Omron CX-Programmer project NewProject (CX-Programmer 9.61)

# PLC NewPLC1: CJ1M CPU11

## Global symbols (name address type ; comment)
0.00 BOOL  ; PB_Start
0.01 BOOL  ; PB_Stop
10.00 BOOL  ; IR_Control
10.01 BOOL  ; SIMPANG 1 = HIJAU
10.02 BOOL  ; SIMPANG 1 = KUNING
10.03 BOOL  ; SIMPANG1 = MERAH
10.04 BOOL  ; SIMPANG 2= HIJAU
10.05 BOOL  ; SIMPANG 2 = KUNING
10.06 BOOL  ; SIMPANG 2 = MERAH
10.07 BOOL  ; SIMPANG 3 = HIJAU
10.08 BOOL  ; SIMPANG 3 = KUNING
10.09 BOOL  ; SIMPANG 3 = MERAH
10.10 BOOL  ; Lampu hijau pejalan kaki 3
10.11 BOOL  ; Lampu Merah pejalan kaki 1
10.12 BOOL  ; Lampu Hijau Pejalan kaki 1
10.13 BOOL  ; Lampu Merah Pejalan Kaki 2
10.14 BOOL  ; Lampu hijau pejalan kaki 2
10.15 BOOL  ; Lampu merah pejalan kaki 3
1.00 BOOL  ; SIMPANG 1 = HIJAU
1.01 BOOL  ; SIMPANG 1 = KUNING
1.02 BOOL  ; SIMPANG 1 = MERAH
1.03 BOOL  ; Lampu  Merah Pejalan Kaki 1
1.04 BOOL  ; Lampu Hijau Pejalan Kaki 1
1.05 BOOL  ; SIMPANG 2 = HIJAU
1.06 BOOL  ; SIMPANG 2 = KUNING
1.07 BOOL  ; SIMPANG 2 = MERAH
1.08 BOOL  ; Lampu Merah Pejalan Kaki 2
1.09 BOOL  ; Lampu Hijau Pejalan Kaki 2
1.10 BOOL  ; SIMPANG 3 = HIJAU
1.11 BOOL  ; SIMPANG 3 = KUNING
1.12 BOOL  ; SIMPANG 3 = MERAH
1.13 BOOL  ; Lampu Merah Pejalan Kaki 3
1.14 BOOL  ; Lampu Hijau Pejalan Kaki 3
1.15 BOOL  ; Lampu Merah Pejalan Kaki 3
200.00 BOOL  ; IR_Control
T0001 BOOL  ; Timer 1
T0002 BOOL  ; Timer 2
T0003 BOOL  ; Timer 3
T0004 BOOL  ; Timer 4
T0005 BOOL  ; Timer 5
T0006 BOOL  ; Timer 6

## Program NewProgram1 (cyclic task 0)

### Section Section1

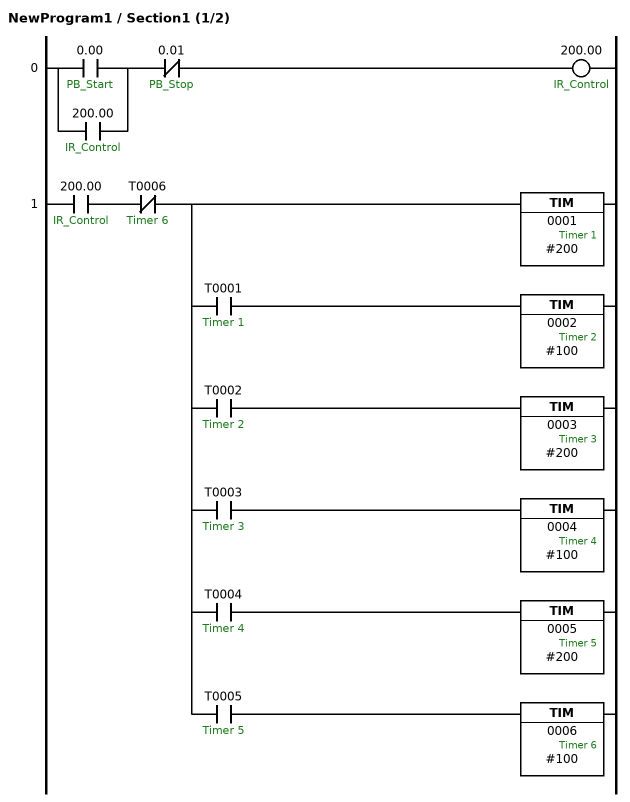
; rung 0
LD 0.00  ; PB_Start
OR 200.00  ; IR_Control
ANDNOT 0.01  ; PB_Stop
OUT 200.00  ; IR_Control
; rung 1
LD 200.00  ; IR_Control
ANDNOT T0006  ; Timer 6
OUT TR0
TIM 0001 #200  ; Timer 1
AND T0001  ; Timer 1
TIM 0002 #100  ; Timer 2
LD TR0
AND T0002  ; Timer 2
TIM 0003 #200  ; Timer 3
LD TR0
AND T0003  ; Timer 3
TIM 0004 #100  ; Timer 4
LD TR0
AND T0004  ; Timer 4
TIM 0005 #200  ; Timer 5
LD TR0
AND T0005  ; Timer 5
TIM 0006 #100  ; Timer 6

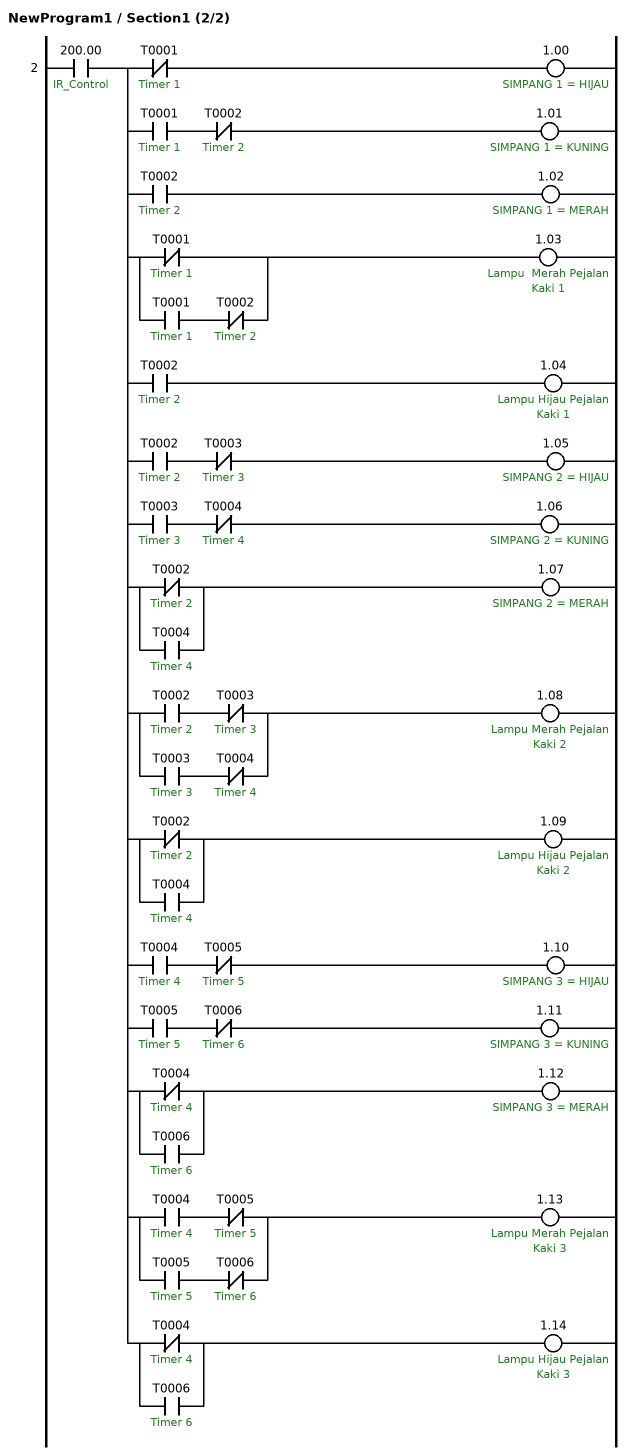
; rung 2
LD 200.00  ; IR_Control
OUT TR0
ANDNOT T0001  ; Timer 1
OUT 1.00  ; SIMPANG 1 = HIJAU
LD TR0
AND T0001  ; Timer 1
ANDNOT T0002  ; Timer 2
OUT 1.01  ; SIMPANG 1 = KUNING
LD TR0
AND T0002  ; Timer 2
OUT 1.02  ; SIMPANG 1 = MERAH
LD TR0
LDNOT T0001  ; Timer 1
LD T0001  ; Timer 1
ANDNOT T0002  ; Timer 2
ORLD
ANDLD
OUT 1.03  ; Lampu  Merah Pejalan Kaki 1
LD TR0
AND T0002  ; Timer 2
OUT 1.04  ; Lampu Hijau Pejalan Kaki 1
LD TR0
AND T0002  ; Timer 2
ANDNOT T0003  ; Timer 3
OUT 1.05  ; SIMPANG 2 = HIJAU
LD TR0
AND T0003  ; Timer 3
ANDNOT T0004  ; Timer 4
OUT 1.06  ; SIMPANG 2 = KUNING
LD TR0
LDNOT T0002  ; Timer 2
OR T0004  ; Timer 4
ANDLD
OUT 1.07  ; SIMPANG 2 = MERAH
LD TR0
LD T0002  ; Timer 2
ANDNOT T0003  ; Timer 3
LD T0003  ; Timer 3
ANDNOT T0004  ; Timer 4
ORLD
ANDLD
OUT 1.08  ; Lampu Merah Pejalan Kaki 2
LD TR0
LDNOT T0002  ; Timer 2
OR T0004  ; Timer 4
ANDLD
OUT 1.09  ; Lampu Hijau Pejalan Kaki 2
LD TR0
AND T0004  ; Timer 4
ANDNOT T0005  ; Timer 5
OUT 1.10  ; SIMPANG 3 = HIJAU
LD TR0
AND T0005  ; Timer 5
ANDNOT T0006  ; Timer 6
OUT 1.11  ; SIMPANG 3 = KUNING
LD TR0
LDNOT T0004  ; Timer 4
OR T0006  ; Timer 6
ANDLD
OUT 1.12  ; SIMPANG 3 = MERAH
LD TR0
LD T0004  ; Timer 4
ANDNOT T0005  ; Timer 5
LD T0005  ; Timer 5
ANDNOT T0006  ; Timer 6
ORLD
ANDLD
OUT 1.13  ; Lampu Merah Pejalan Kaki 3
LD TR0
LDNOT T0004  ; Timer 4
OR T0006  ; Timer 6
ANDLD
OUT 1.14  ; Lampu Hijau Pejalan Kaki 3

### Section END
; rung 0
END(001)